# EPICS substitutions: db/ecmcEL5021.substitutions
# All fields related to postion scaling and alarms
file ecmcEL5021.template
{
	pattern {LINR,    ESLO,   EOFF,   EGU,        PREC, LOW, LOLO, HIGH, HIHI, HYST, LLSV,       LSV,        HSV,        HHSV      }
		{"SLOPE", 1,      0,      "Steps",    0,    0,   0,    0,    0,    0,    "NO_ALARM", "NO_ALARM", "NO_ALARM", "NO_ALARM"}
}
